FUNCTION_BLOCK FB_Toggle
VAR_INPUT
	CLK : BOOL;
END_VAR
VAR_OUTPUT
	Q : BOOL;
END_VAR
VAR
	s_osr : R_TRIG;
END_VAR


s_osr(CLK := CLK);

IF s_osr.Q AND Q THEN
	Q := FALSE; 
ELSIF s_osr.Q AND NOT(Q) THEN	
	Q := TRUE;
END_IF

END_FUNCTION_BLOCK

(* stored: Version 1.1.0.1, ProductVersion 3.1.4024.12
   POU FB_Toggle: Id {bc3b0774-fe4f-4cbd-a043-08f9c1e5a0d2}, SpecialFunc None *)
